TYPE ST_SensorValues :
STRUCT

END_STRUCT
END_TYPE

(* stored: Version 1.1.0.1, ProductVersion 3.1.4024.12
   DUT ST_SensorValues: Id {3b9d9001-2ea4-4898-9ddf-20f3934c3003} *)
